// Mitsubishi GX Works2 project: 김건태   PLC: Q02/Q02H

PROGRAM PLC
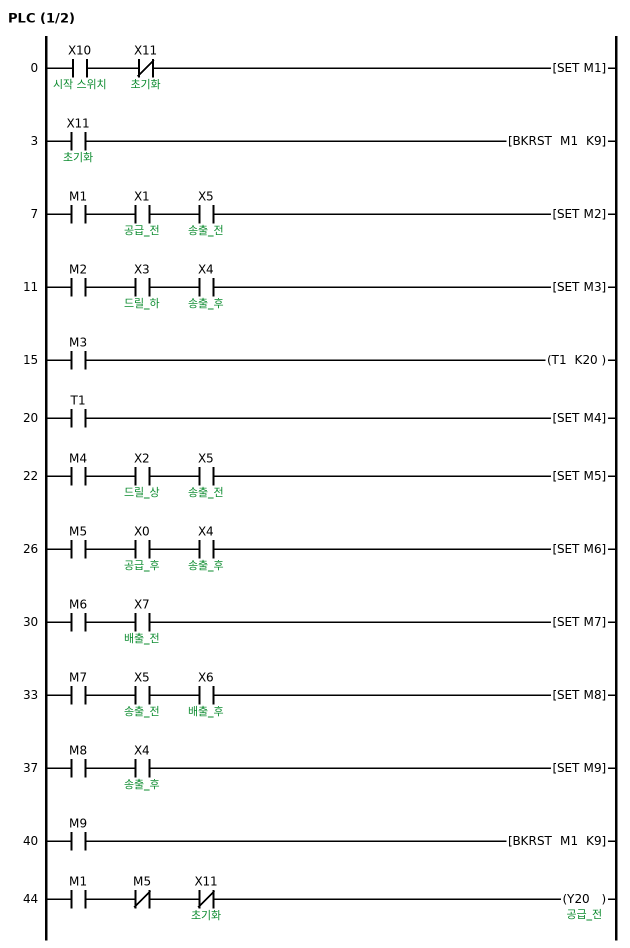
0     LD      X10  ; 시작 스위치
      ANI     X11  ; 초기화
      SET     M1
3     LD      X11  ; 초기화
      BKRST   M1 K9
7     LD      M1
      AND     X1  ; 공급_전
      AND     X5  ; 송출_전
      SET     M2
11    LD      M2
      AND     X3  ; 드릴_하
      AND     X4  ; 송출_후
      SET     M3
15    LD      M3
      OUT     T1 K20
20    LD      T1
      SET     M4
22    LD      M4
      AND     X2  ; 드릴_상
      AND     X5  ; 송출_전
      SET     M5
26    LD      M5
      AND     X0  ; 공급_후
      AND     X4  ; 송출_후
      SET     M6
30    LD      M6
      AND     X7  ; 배출_전
      SET     M7
33    LD      M7
      AND     X5  ; 송출_전
      AND     X6  ; 배출_후
      SET     M8
37    LD      M8
      AND     X4  ; 송출_후
      SET     M9
40    LD      M9
      BKRST   M1 K9
44    LD      M1
      ANI     M5
      ANI     X11  ; 초기화
      OUT     Y20  ; 공급_전
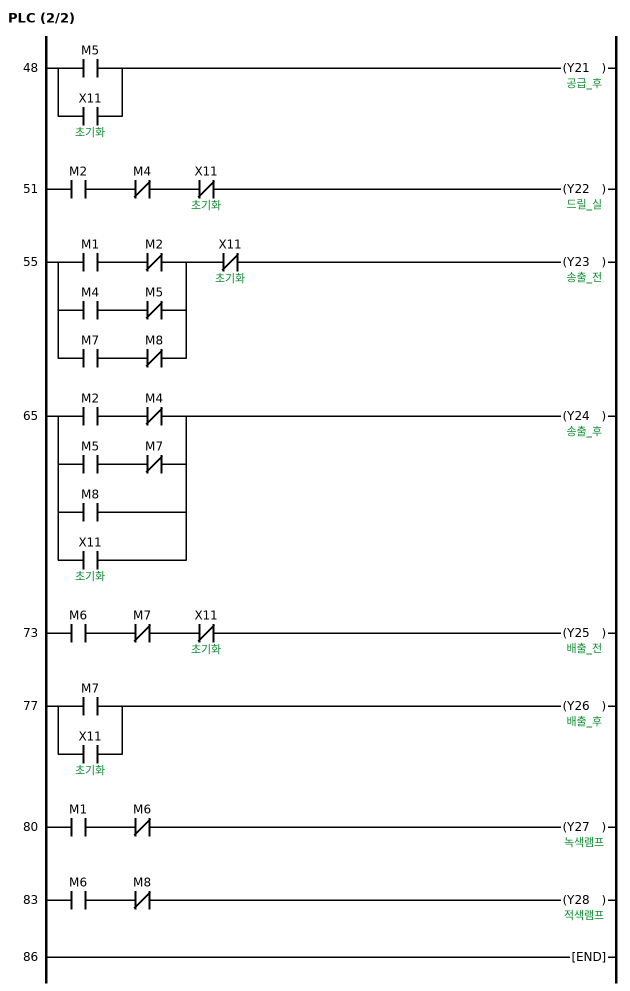
48    LD      M5
      OR      X11  ; 초기화
      OUT     Y21  ; 공급_후
51    LD      M2
      ANI     M4
      ANI     X11  ; 초기화
      OUT     Y22  ; 드릴_실
55    LD      M1
      ANI     M2
      LD      M4
      ANI     M5
      ORB
      LD      M7
      ANI     M8
      ORB
      ANI     X11  ; 초기화
      OUT     Y23  ; 송출_전
65    LD      M2
      ANI     M4
      LD      M5
      ANI     M7
      ORB
      OR      M8
      OR      X11  ; 초기화
      OUT     Y24  ; 송출_후
73    LD      M6
      ANI     M7
      ANI     X11  ; 초기화
      OUT     Y25  ; 배출_전
77    LD      M7
      OR      X11  ; 초기화
      OUT     Y26  ; 배출_후
80    LD      M1
      ANI     M6
      OUT     Y27  ; 녹색램프
83    LD      M6
      ANI     M8
      OUT     Y28  ; 적색램프
86    END
END_PROGRAM

PROGRAM HMI
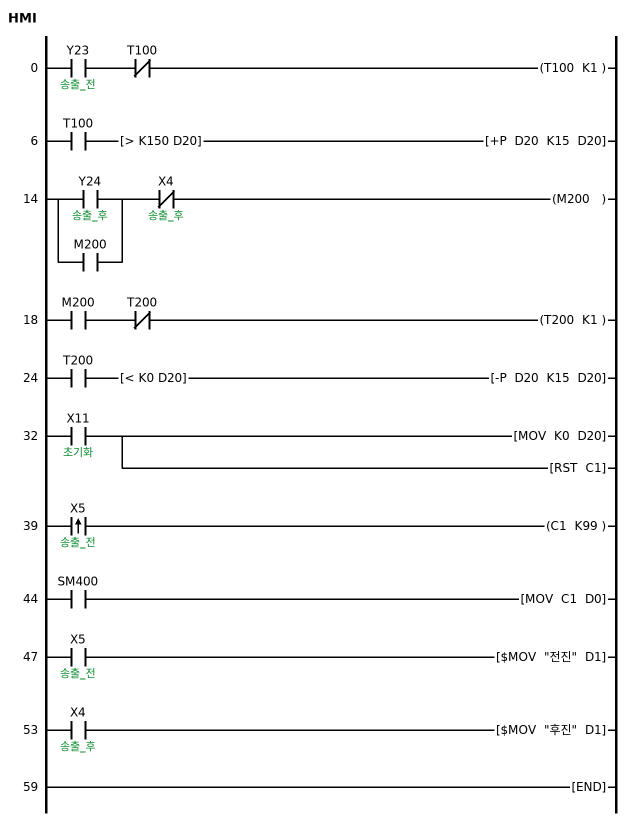
0     LD      Y23  ; 송출_전
      ANI     T100
      OUT     T100 K1
6     LD      T100
      AND>    K150 D20
      +P      D20 K15 D20
14    LD      Y24  ; 송출_후
      OR      M200
      ANI     X4  ; 송출_후
      OUT     M200
18    LD      M200
      ANI     T200
      OUT     T200 K1
24    LD      T200
      AND<    K0 D20
      -P      D20 K15 D20
32    LD      X11  ; 초기화
      MOV     K0 D20
      RST     C1
39    LDP     X5  ; 송출_전
      OUT     C1 K99
44    LD      SM400
      MOV     C1 D0
47    LD      X5  ; 송출_전
      $MOV    "전진" D1
53    LD      X4  ; 송출_후
      $MOV    "후진" D1
59    END
END_PROGRAM
